SUBAPPLICATION Ventilsteuerung_Uebung_002 (* DigitalInput_I1 auf DigitalOutput_Q1 *)
  (* Standard: 61499-2 *)
  (* Version 1.0, 2023-10-23, franz *)
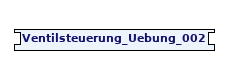
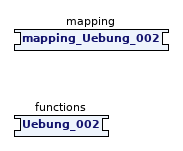
  SUBAPPS
    mapping : mapping_Uebung_002;
    functions : Uebung_002;
  END_SUBAPPS
END_SUBAPPLICATION
